Staubli VAL3: push.pgx

public program push(MotionBuffer& x_cmd, bool& x_res)
begin
  if (nElems < size(buffer))
    buffer[nPush] = x_cmd
    nElems = nElems + 1
    nPush = nPush + 1
    if (nPush >= size(buffer))
      nPush = 0
    endIf
    x_res = true
  else
    x_res = false
  endIf
end
